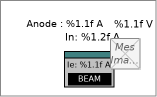
VISUALIZATION VISU_MARK3_PLUS_COTE  // 157x97
VAR_IN_OUT
	m_Input_IAD : BLOCK_MARK3_PLUS;
END_VAR
    Polygon (59,48), invisible if: NOT m_Input_IAD.STATE_BEAM_ON
    Polygon (91,50), invisible if: NOT m_Input_IAD.STATE_BEAM_ON
    Polygon (86,81)
    Rectangle (85,69 25x10), "ON"
    RoundedRectangle (64,51 50x36)
    Rectangle (64,51 50x7)
    RoundedRectangle (68,73 43x12), "BEAM", colour toggle: (m_Input_IAD.STATE_BEAM_ON) <> 0
    Rectangle (51,58 76x14), "Ie: %1.1f A", text variable: m_Input_IAD.STATE_I_Emi, invisible if: NOT m_Input_IAD.STATE_BEAM
    Rectangle (63,52 52x32), input disabled if: ((NOT m_Input_IAD.BEAM.AUTOR_ON_IHM AND NOT m_Input_IAD.BEAM.AUTOR_OFF_IHM) OR NOT PRG_User.ACTU_USER.MAINTENANCE) <> 0
        OnMouseUp: execute { m_Input_IAD.BEAM.M_On:=(TRUE); }
    RoundedRectangle (68,73 43x12), "BEAM", invisible if: (m_Input_IAD.STATE_BEAM_ON OR m_Input_IAD.STATE_BEAM) <> 0
    Rectangle (25,17 83x14), "Anode : %1.1f A", text variable: m_Input_IAD.STATE_I_Anode, invisible if: NOT m_Input_IAD.STATE_BEAM
    Rectangle (107,17 50x14), "%1.1f V", text variable: m_Input_IAD.STATE_V_Anode, invisible if: NOT m_Input_IAD.STATE_BEAM
    Rectangle (60,30 62x14), "In: %1.2f A", text variable: m_Input_IAD.STATE_I_Neut, invisible if: NOT m_Input_IAD.STATE_BEAM
    Polygon (47,55)
    Image (110,38 30x31), invisible if: NOT m_Input_IAD.STATE_Nok, image: MesImages.warning
END_VISUALIZATION

(* stored: Version 1.1.0.1, ProductVersion 3.1.4024.10
   Visu VISU_MARK3_PLUS_COTE: Id {c7dfdc91-32d0-471c-a902-e40c5f383b5d} *)
